Staubli VAL3: setAnaValue.pgx

public program setAnaValue(num x_nValue, string x_sItem)
begin
  // set the value in to the AIO
  aioSet(saveInOut:aOutput[x_sItem].aAio,x_nValue)
end
